// TIA Portal V18 export
// export: Created 2025-12-01T12:39:35.7627715Z, ExportSetting None, DisplayName Totally Integrated Automation Portal, DisplayVersion V18 Update 5, DisplayName TIA Portal Openness, DisplayVersion V18 Update 5, DisplayName TIA Portal Teamcenter Gateway, DisplayVersion V18, DisplayName TIA Portal Version Control Interface, DisplayVersion V18, DisplayName STEP 7 Professional, DisplayVersion V18 Update 5, DisplayName STEP 7 Safety, DisplayVersion V18, DisplayName WinCC Professional, DisplayVersion V18 Update 5
VAR_GLOBAL   // PLC tag table "TestResult"
END_VAR
VAR_GLOBAL CONSTANT   // user constants
   VacuumTestOK : Int := 1;
   VacuumTestNG : Int := 2;
   NitTestNG : Int := 2;
   NitTestOK : Int := 1;
END_VAR
